PROGRAM MAIN
VAR
END_VAR

END_PROGRAM

(* stored: Version 1.1.0.1
   POU MAIN: Id {b2020ea4-8f51-4aab-baa8-76b366a6a555} *)
